FUNCTION_BLOCK AQ_SPLIT_8 (* Fan-Out: Splits 1 AQ into 8 AQ adapters *)
  (* Standard: 61499-2; Description: Copyright (c) 2026 Meisterschulen am Ostbahnhof SPDX-License-Identifier: EPL-2.0 *)
  (* Version 1.0, 2026-05-16, Franz Höpfinger, Meisterschulen am Ostbahnhof, Initial Version *)
  PACKAGE adapter::events::unidirectional;
  IMPORT eclipse4diac::core::GenericClassName;
  {SET_ATTRIBUTE(eclipse4diac::core::GenericClassName, 'GEN_AQ_SPLIT')}
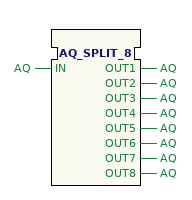
  SOCKETS
    IN : adapter::types::unidirectional::AQ;
  END_SOCKETS
  PLUGS
    OUT1 : adapter::types::unidirectional::AQ;
    OUT2 : adapter::types::unidirectional::AQ;
    OUT3 : adapter::types::unidirectional::AQ;
    OUT4 : adapter::types::unidirectional::AQ;
    OUT5 : adapter::types::unidirectional::AQ;
    OUT6 : adapter::types::unidirectional::AQ;
    OUT7 : adapter::types::unidirectional::AQ;
    OUT8 : adapter::types::unidirectional::AQ;
  END_PLUGS
END_FUNCTION_BLOCK
